// TIA Portal V20 export
VAR_GLOBAL   // PLC tag table "Safety_Drive"
   Axis01_X_Status AT %I6812.0 : "LDrvSafe_typeSinaTlg903Status";
   Axis02_Y_Status AT %I6828.0 : "LDrvSafe_typeSinaTlg903Status";
   Axis03_ZM_Status AT %I6844.0 : "LDrvSafe_typeSinaTlg903Status";
   Axis04_B_Status AT %I6764.0 : "LDrvSafe_typeSinaTlg903Status";
   Axis05_U1_Status AT %I6700.0 : "LDrvSafe_typeSinaTlg903Status";
   Axis06_U2_Status AT %I6748.0 : "LDrvSafe_typeSinaTlg903Status";
   Axis07_V_Status AT %I6716.0 : "LDrvSafe_typeSinaTlg903Status";
   Axis08_W_Status AT %I6732.0 : "LDrvSafe_typeSinaTlg903Status";
   Axis09_ZL_Status AT %I6860.0 : "LDrvSafe_typeSinaTlg903Status";
   Axis01_X_Control AT %Q6812.0 : "LDrvSafe_typeSinaTlg903Control";
   Axis02_Y_Control AT %Q6828.0 : "LDrvSafe_typeSinaTlg903Control";
   Axis03_ZM_Control AT %Q6844.0 : "LDrvSafe_typeSinaTlg903Control";
   Axis04_B_Control AT %Q6764.0 : "LDrvSafe_typeSinaTlg903Control";
   Axis05_U1_Control AT %Q6700.0 : "LDrvSafe_typeSinaTlg903Control";
   Axis06_U2_Control AT %Q6748.0 : "LDrvSafe_typeSinaTlg903Control";
   Axis07_V_Control AT %Q6716.0 : "LDrvSafe_typeSinaTlg903Control";
   Axis08_W_Control AT %Q6732.0 : "LDrvSafe_typeSinaTlg903Control";
   Axis09_ZL_Control AT %Q6860.0 : "LDrvSafe_typeSinaTlg903Control";
END_VAR
